// SIMATIC S7-200 project (STEP 7-Micro/WIN), CPU 221 REL 01.10

SYMBOL_TABLE IO
I急停按钮            I0.0
I复位按钮            I0.1
I自动/手动           I0.2
I启动按钮1           I0.3
I启动按钮2           I0.4
I安全光幕            I0.5
I增压缸原位           I1.0
I增压缸进位           I1.1
I顶升气缸下降          I1.3
I顶升气缸顶升          I1.4
Q增压气缸泄压          Q0.4
Q增压气缸增压          Q0.5
Q增压气缸下降          Q0.6
Q增压气缸上升          Q0.7
Q顶升气缸下降          Q1.0
Q顶升气缸顶升          Q1.1
红灯               Q2.0
绿灯               Q2.1
黄灯               Q2.2
蜂鸣器              Q2.3
END_SYMBOL_TABLE

SYMBOL_TABLE M3000
流水线工步号           MW3000
压装自动工步号          MW3004
芯片编号             MW3006
通讯状态             M3010.0
本工位合格            M3010.1
本工位完成            M3010.2
不合格报警            M3010.3
RFID读取触发         M3010.4
RFID读取完成         M3010.5
RFID运行中          M3010.6
M一键初始化按钮         M3011.0
M一键初始化完成         M3011.1
M增压缸下降           M3021.0
M增压缸上升           M3021.1
M增压缸增压           M3021.2
M增压缸泄压           M3021.3
M顶转向器气缸顶升        M3021.4
M顶转向器气缸下降        M3021.5
上工位合格            M3030.0
上工位完成            M3030.1
联线状态             M3040.0
报警工步号            MW3050
员工权限             M3060.0
END_SYMBOL_TABLE
